FUNCTION_BLOCK FB_Datalogger_SENECA EXTENDS FB_Datalogger_Base
 

VAR_INPUT PERSISTENT
	ParamWriteTimeout			: TIME  	:= T#5S ;		  					(* (Time) Timeout for modbus reading*)
END_VAR

       	
VAR_INPUT           	
	// I/O Inputs 
	
END_VAR             	
      	
VAR 
MesDataExd				: Datalogger_SENECA;                		
	
//INPUT Modbus
	FB_ModbusRead	          	: ARRAY[1..2] OF FB_ModbusRead; 	            // (NA) FB for Modbus Reading	
	MesBlock1_Temp				: ARRAY [1..8] OF WORD ; 
	
	AlarmModbusInput			: BOOL;
	AlarmID_ModbusInput			: UDINT;
END_VAR

METHOD M_Execute : BOOL
VAR_INPUT
END_VAR

		MesDataExd.MesData.MesWindSp := 14;
		MesDataExd.MesWindDir := 80;
END_METHOD

END_FUNCTION_BLOCK

(* stored: Version 1.1.0.1, ProductVersion 3.1.4024.9
   POU FB_Datalogger_SENECA: Id {fb95c73f-0b84-438b-a7a8-699e8ea07c46}, SpecialFunc None
   Method M_Execute: Id {ea5cf854-5e24-4528-8f3c-4a96b530c3d1} *)
